# EPICS substitutions: BLDApp/Db/eOrbitsFcomHXR.substitutions
file eOrbitsFcom.substitutions
{
  pattern
  { BPM1, BPM2, BPM3, BPM4, BPM5, BPM6, BPM7, BPM8, BPM9, BPM10, BPM11, EC }
  { BPMS:LTUH:910:, BPMS:LTUH:960:, BPMS:UNDH:1305:, BPMS:UNDH:1390:, BPMS:UNDH:1490:, BPMS:UNDH:1590:, BPMS:UNDH:1690:, BPMS:UNDH:1790:, BPMS:UNDH:1890:, BPMS:UNDH:1990:, BPMS:UNDH:2090:, $(EC)}

}
